{attribute 'qualified_only'}
{attribute 'to_string'}
TYPE E_ControllerArmStates :
(
	Idle:=0,
	Selftest1,
	Selftest2,
	Ergonomics1,
	Ergonomics2,
	Teleoperation1
)UINT := Idle
;
END_TYPE

(* stored: Version 1.1.0.1, ProductVersion 3.1.4024.12
   EnumerationTextList E_ControllerArmStates: Id {a676d58d-ed6e-46c3-a33a-24142845b7c3} *)
